INTERFACE I_AsyncStatus

PROPERTY Busy : bool
GET
END_GET
END_PROPERTY

PROPERTY Done : bool
GET
END_GET
END_PROPERTY

PROPERTY Error : bool
GET
END_GET
END_PROPERTY

END_INTERFACE

(* stored: Version 1.1.0.1, ProductVersion 3.1.4024.3
   Itf I_AsyncStatus: Id {b3a2d6a6-21d0-4b08-be03-157cda3ff6a5}
   Property Busy: Id {1c66b9e6-2211-46e3-ba02-f7b107e3230e}
   Get Get: Id {01ffbed5-9871-4b26-a05d-34e8042ca539}
   Property Done: Id {3558482a-dd8d-4732-8d58-fc73394ccb24}
   Get Get: Id {8bd8b890-d718-4598-b904-0b2c09e43069}
   Property Error: Id {575b3820-40ec-432c-ac3e-c18c7478061e}
   Get Get: Id {0d9cb2b3-d0a9-46be-8d7d-a6a0c3cdff4e} *)
